DATA_BLOCK "CALHA VIBRATÓRIA_DB"
{ S7_Optimized_Access := 'TRUE' }
VERSION : 0.1
NON_RETAIN
"CALHA VIBRATÓRIA"

BEGIN

END_DATA_BLOCK

